// TIA Portal V19 export
FUNCTION "FC30_FerRobotic" : Void   // FC30, LAD
TITLE = FerRobotic communication
{ S7_Optimized_Access := 'TRUE' }
// stored: AutoNumber false, IsIECCheckEnabled true, SetENOAutomatically false
BEGIN

REGION Network 1: Swap byte of value to Receive from FerRobotic
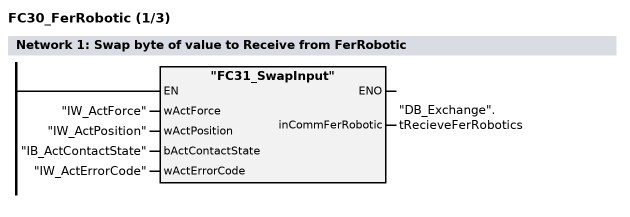
   RUNG wire#powerrail
      "FC31_SwapInput"(wActForce := "IW_ActForce", wActPosition := "IW_ActPosition", bActContactState := "IB_ActContactState", wActErrorCode := "IW_ActErrorCode", inCommFerRobotic => "DB_Exchange".tRecieveFerRobotics)
   END_RUNG
   // the same network as SCL:
   "FC31_SwapInput"(wActForce := "IW_ActForce",
                    wActPosition := "IW_ActPosition",
                    bActContactState := "IB_ActContactState",
                    wActErrorCode := "IW_ActErrorCode",
                    inCommFerRobotic => "DB_Exchange".tRecieveFerRobotics);
END_REGION

REGION Network 2: Comminucation with FerRobotic System
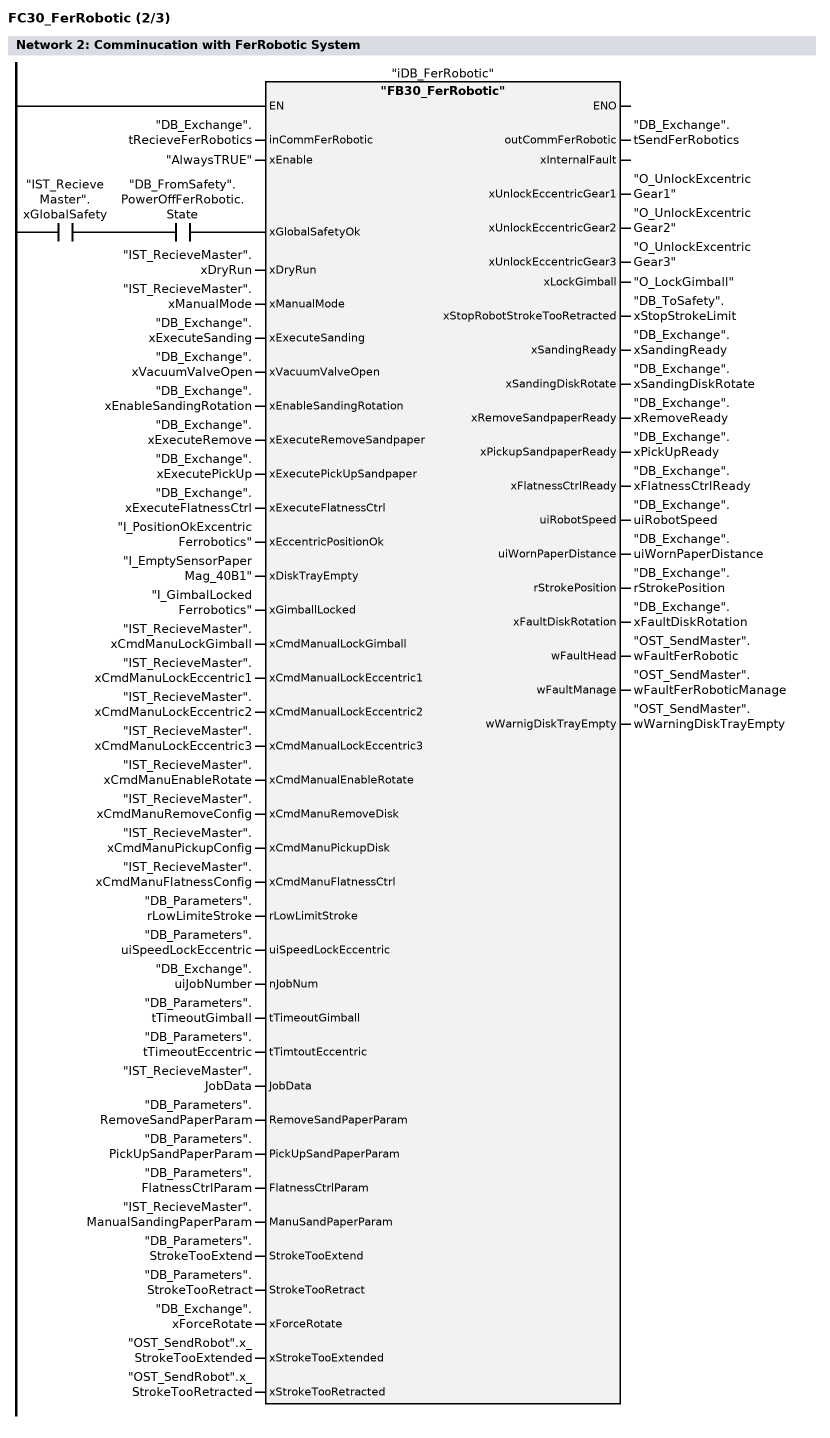
   RUNG wire#powerrail
      "iDB_FerRobotic"(xGlobalSafetyOk := wire#w1, inCommFerRobotic := "DB_Exchange".tRecieveFerRobotics, xEnable := "AlwaysTRUE", xDryRun := "IST_RecieveMaster".xDryRun, xManualMode := "IST_RecieveMaster".xManualMode, xExecuteSanding := "DB_Exchange".xExecuteSanding, xVacuumValveOpen := "DB_Exchange".xVacuumValveOpen, xEnableSandingRotation := "DB_Exchange".xEnableSandingRotation, xExecuteRemoveSandpaper := "DB_Exchange".xExecuteRemove, xExecutePickUpSandpaper := "DB_Exchange".xExecutePickUp, xExecuteFlatnessCtrl := "DB_Exchange".xExecuteFlatnessCtrl, xEccentricPositionOk := "I_PositionOkExcentricFerrobotics", xDiskTrayEmpty := "I_EmptySensorPaperMag_40B1", xGimballLocked := "I_GimbalLockedFerrobotics", xCmdManualLockGimball := "IST_RecieveMaster".xCmdManuLockGimball, xCmdManualLockEccentric1 := "IST_RecieveMaster".xCmdManuLockEccentric1, xCmdManualLockEccentric2 := "IST_RecieveMaster".xCmdManuLockEccentric2, xCmdManualLockEccentric3 := "IST_RecieveMaster".xCmdManuLockEccentric3, xCmdManualEnableRotate := "IST_RecieveMaster".xCmdManuEnableRotate, xCmdManuRemoveDisk := "IST_RecieveMaster".xCmdManuRemoveConfig, xCmdManuPickupDisk := "IST_RecieveMaster".xCmdManuPickupConfig, xCmdManuFlatnessCtrl := "IST_RecieveMaster".xCmdManuFlatnessConfig, rLowLimitStroke := "DB_Parameters".rLowLimiteStroke, uiSpeedLockEccentric := "DB_Parameters".uiSpeedLockEccentric, nJobNum := "DB_Exchange".uiJobNumber, tTimeoutGimball := "DB_Parameters".tTimeoutGimball, tTimtoutEccentric := "DB_Parameters".tTimeoutEccentric, JobData := "IST_RecieveMaster".JobData, RemoveSandPaperParam := "DB_Parameters".RemoveSandPaperParam, PickUpSandPaperParam := "DB_Parameters".PickUpSandPaperParam, FlatnessCtrlParam := "DB_Parameters".FlatnessCtrlParam, ManuSandPaperParam := "IST_RecieveMaster".ManualSandingPaperParam, StrokeTooExtend := "DB_Parameters".StrokeTooExtend, StrokeTooRetract := "DB_Parameters".StrokeTooRetract, xForceRotate := "DB_Exchange".xForceRotate, xStrokeTooExtended := "OST_SendRobot".x_StrokeTooExtended, xStrokeTooRetracted := "OST_SendRobot".x_StrokeTooRetracted, outCommFerRobotic => "DB_Exchange".tSendFerRobotics, xInternalFault =>, xUnlockEccentricGear1 => "O_UnlockExcentricGear1", xUnlockEccentricGear2 => "O_UnlockExcentricGear2", xUnlockEccentricGear3 => "O_UnlockExcentricGear3", xLockGimball => "O_LockGimball", xStopRobotStrokeTooRetracted => "DB_ToSafety".xStopStrokeLimit, xSandingReady => "DB_Exchange".xSandingReady, xSandingDiskRotate => "DB_Exchange".xSandingDiskRotate, xRemoveSandpaperReady => "DB_Exchange".xRemoveReady, xPickupSandpaperReady => "DB_Exchange".xPickUpReady, xFlatnessCtrlReady => "DB_Exchange".xFlatnessCtrlReady, uiRobotSpeed => "DB_Exchange".uiRobotSpeed, uiWornPaperDistance => "DB_Exchange".uiWornPaperDistance, rStrokePosition => "DB_Exchange".rStrokePosition, xFaultDiskRotation => "DB_Exchange".xFaultDiskRotation, wFaultHead => "OST_SendMaster".wFaultFerRobotic, wFaultManage => "OST_SendMaster".wFaultFerRoboticManage, wWarnigDiskTrayEmpty => "OST_SendMaster".wWarningDiskTrayEmpty)
   END_RUNG
   RUNG wire#powerrail
      Contact( "IST_RecieveMaster".xGlobalSafety )
      Contact( "DB_FromSafety".PowerOffFerRobotic.State )
   END_RUNG wire#w1
   // the same network as SCL:
   "iDB_FerRobotic"(inCommFerRobotic := "DB_Exchange".tRecieveFerRobotics,   // "FB30_FerRobotic"
                    xEnable := "AlwaysTRUE",
                    xGlobalSafetyOk := "IST_RecieveMaster".xGlobalSafety AND "DB_FromSafety".PowerOffFerRobotic.State,
                    xDryRun := "IST_RecieveMaster".xDryRun,
                    xManualMode := "IST_RecieveMaster".xManualMode,
                    xExecuteSanding := "DB_Exchange".xExecuteSanding,
                    xVacuumValveOpen := "DB_Exchange".xVacuumValveOpen,
                    xEnableSandingRotation := "DB_Exchange".xEnableSandingRotation,
                    xExecuteRemoveSandpaper := "DB_Exchange".xExecuteRemove,
                    xExecutePickUpSandpaper := "DB_Exchange".xExecutePickUp,
                    xExecuteFlatnessCtrl := "DB_Exchange".xExecuteFlatnessCtrl,
                    xEccentricPositionOk := "I_PositionOkExcentricFerrobotics",
                    xDiskTrayEmpty := "I_EmptySensorPaperMag_40B1",
                    xGimballLocked := "I_GimbalLockedFerrobotics",
                    xCmdManualLockGimball := "IST_RecieveMaster".xCmdManuLockGimball,
                    xCmdManualLockEccentric1 := "IST_RecieveMaster".xCmdManuLockEccentric1,
                    xCmdManualLockEccentric2 := "IST_RecieveMaster".xCmdManuLockEccentric2,
                    xCmdManualLockEccentric3 := "IST_RecieveMaster".xCmdManuLockEccentric3,
                    xCmdManualEnableRotate := "IST_RecieveMaster".xCmdManuEnableRotate,
                    xCmdManuRemoveDisk := "IST_RecieveMaster".xCmdManuRemoveConfig,
                    xCmdManuPickupDisk := "IST_RecieveMaster".xCmdManuPickupConfig,
                    xCmdManuFlatnessCtrl := "IST_RecieveMaster".xCmdManuFlatnessConfig,
                    rLowLimitStroke := "DB_Parameters".rLowLimiteStroke,
                    uiSpeedLockEccentric := "DB_Parameters".uiSpeedLockEccentric,
                    nJobNum := "DB_Exchange".uiJobNumber,
                    tTimeoutGimball := "DB_Parameters".tTimeoutGimball,
                    tTimtoutEccentric := "DB_Parameters".tTimeoutEccentric,
                    JobData := "IST_RecieveMaster".JobData,
                    RemoveSandPaperParam := "DB_Parameters".RemoveSandPaperParam,
                    PickUpSandPaperParam := "DB_Parameters".PickUpSandPaperParam,
                    FlatnessCtrlParam := "DB_Parameters".FlatnessCtrlParam,
                    ManuSandPaperParam := "IST_RecieveMaster".ManualSandingPaperParam,
                    StrokeTooExtend := "DB_Parameters".StrokeTooExtend,
                    StrokeTooRetract := "DB_Parameters".StrokeTooRetract,
                    xForceRotate := "DB_Exchange".xForceRotate,
                    xStrokeTooExtended := "OST_SendRobot".x_StrokeTooExtended,
                    xStrokeTooRetracted := "OST_SendRobot".x_StrokeTooRetracted,
                    outCommFerRobotic => "DB_Exchange".tSendFerRobotics,
                    xUnlockEccentricGear1 => "O_UnlockExcentricGear1",
                    xUnlockEccentricGear2 => "O_UnlockExcentricGear2",
                    xUnlockEccentricGear3 => "O_UnlockExcentricGear3",
                    xLockGimball => "O_LockGimball",
                    xStopRobotStrokeTooRetracted => "DB_ToSafety".xStopStrokeLimit,
                    xSandingReady => "DB_Exchange".xSandingReady,
                    xSandingDiskRotate => "DB_Exchange".xSandingDiskRotate,
                    xRemoveSandpaperReady => "DB_Exchange".xRemoveReady,
                    xPickupSandpaperReady => "DB_Exchange".xPickUpReady,
                    xFlatnessCtrlReady => "DB_Exchange".xFlatnessCtrlReady,
                    uiRobotSpeed => "DB_Exchange".uiRobotSpeed,
                    uiWornPaperDistance => "DB_Exchange".uiWornPaperDistance,
                    rStrokePosition => "DB_Exchange".rStrokePosition,
                    xFaultDiskRotation => "DB_Exchange".xFaultDiskRotation,
                    wFaultHead => "OST_SendMaster".wFaultFerRobotic,
                    wFaultManage => "OST_SendMaster".wFaultFerRoboticManage,
                    wWarnigDiskTrayEmpty => "OST_SendMaster".wWarningDiskTrayEmpty);
END_REGION

REGION Network 3: Swap byte of value to send to FerRobotic
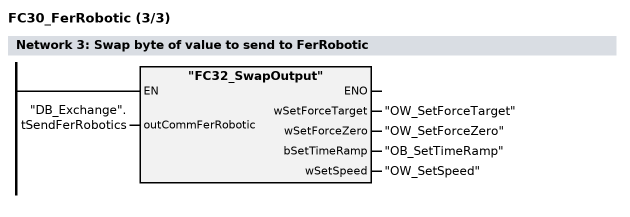
   RUNG wire#powerrail
      "FC32_SwapOutput"(outCommFerRobotic := "DB_Exchange".tSendFerRobotics, wSetForceTarget => "OW_SetForceTarget", wSetForceZero => "OW_SetForceZero", bSetTimeRamp => "OB_SetTimeRamp", wSetSpeed => "OW_SetSpeed")
   END_RUNG
   // the same network as SCL:
   "FC32_SwapOutput"(outCommFerRobotic := "DB_Exchange".tSendFerRobotics,
                     wSetForceTarget => "OW_SetForceTarget",
                     wSetForceZero => "OW_SetForceZero",
                     bSetTimeRamp => "OB_SetTimeRamp",
                     wSetSpeed => "OW_SetSpeed");
END_REGION
END_FUNCTION
